FUNCTION_BLOCK myVeryFirstTcoContext EXTENDS TcoCore.TcoContext
VAR
    {attribute addProperty Name "<#Enter user friendly name of this instance here!!!#>"}
    myVeryFirstDataman : TcoCognexVision.TcoDataman_v_5_x_x(THIS^);
END_VAR

(*~
    <docu>
        <summary>
            Main method of the TcoContext. This is the entry point of any control logic that belongs to this context.
            The call of this method is ensured by calling the <c>InstanceName.Run()</c> method, and it must not be called explicitly.
            This method is abstract, and it must be overridden in derived block.
        </summary>
    </docu>
~*)
METHOD PROTECTED Main
myVeryFirstDataman(inoIoData := GVL.myVeryFirstDatamanGVL);
myVeryFirstDataman.Service();
END_METHOD

END_FUNCTION_BLOCK

(* stored: Version 1.1.0.1, ProductVersion 3.1.4024.11
   POU myVeryFirstTcoContext: Id {c146fb1f-4e72-0d7a-1a50-119df53cfd0b}, SpecialFunc None
   Method Main: Id {d77a27d5-4977-0441-25c3-b6c97ee73678} *)
